// TwinCAT 3 PLC project SQLDemo
// ProgramVersion: 3.1.4026.22
// libraries:
//   Tc2_Standard, * (Beckhoff Automation GmbH)
//   Tc2_System, * (Beckhoff Automation GmbH)
//   Tc2_Utilities, * (Beckhoff Automation GmbH)
//   Tc3_Database, * (Beckhoff Automation GmbH)
//   Tc3_EventLogger, * (Beckhoff Automation GmbH)
// project tree:
//   DUTs/ ST_DbRecord.TcDUT
//   GVLs/ GVL_DB.TcGVL
//   / PlcTask.TcTTO
//   POUs/ FB_SqlLogger.TcPOU, MAIN.TcPOU
// real-time tasks:
//   TASK PlcTask: cycle T#10ms, priority 20, ADS port 350

CONFIGURATION SQLDemo
    RESOURCE PLC ON TwinCAT3
        TASK PlcTask(INTERVAL := T#10ms, PRIORITY := 21);
        PROGRAM MAIN WITH PlcTask : MAIN;
    END_RESOURCE
END_CONFIGURATION

// ---- DUTs/ST_DbRecord.TcDUT
// One row returned by a SELECT from the ds table
TYPE ST_DbRecord : STRUCT
  id        : DINT;
  timestamp : DT;
  value     : REAL;
END_STRUCT
END_TYPE

// ---- GVLs/GVL_DB.TcGVL
{attribute 'qualified_only'}
VAR_GLOBAL CONSTANT
  // Must match the hDBID configured in the TwinCAT Database Server (TF6420)
  DB_ID           : UDINT := 1;
  C_MaxSelectRows : UDINT := 1000;
END_VAR
VAR_GLOBAL
  arrResults   : ARRAY[1..1000] OF ST_DbRecord;
  nResultCount : UDINT;
  bWriteError  : BOOL;
END_VAR

// ---- POUs/MAIN.TcPOU
PROGRAM MAIN
VAR
  // --- System time (used by every FB_SqlLogger) ---
  fbLocalSystemTime : FB_LocalSystemTime;

  // --- Sensor values: replace these with your real signal variables ---
  rTemperature : REAL := 22.5;   // id=1
  rHumidity    : REAL := 55.0;   // id=2
  rSpeed       : REAL := 1450.0; // id=3

  // --- One logger per channel ---
  fbLogTemp  : FB_SqlLogger;
  fbLogHumid : FB_SqlLogger;
  fbLogSpeed : FB_SqlLogger;

  // --- Read back: set bSelect := TRUE to fetch the last 1000 rows ---
  fbSelectDb     : FB_SQLDatabaseEvt(sNetID := '', tTimeout := T#30S);
  fbSelectCmd    : FB_SQLCommandEvt(sNetID := '', tTimeout := T#30S);
  fbSelectResult : FB_SQLResultEvt(sNetID := '', tTimeout := T#30S);
  sSelectCmd     : STRING(255) := 'SELECT id, timestamp, value FROM ds ORDER BY timestamp DESC LIMIT 1000';
  bSelect        : BOOL;
  bSelectBusy    : BOOL;
  bSelectError   : BOOL;
  nSelectState   : INT; // 0=idle,1=connect,2=createCmd,3=execute,4=read,5=disconnect
  ipSelectResult : Tc3_EventLogger.I_TcMessage;
END_VAR

// --- System time ---
fbLocalSystemTime(bEnable := TRUE);

// --- Write: log each channel on its own interval ---
fbLogTemp(
  id           := 1,
  rValue       := rTemperature,
  nIntervalSec := 10,
  nDbHandle    := GVL_DB.DB_ID,
  stSystemTime := fbLocalSystemTime.systemTime);

fbLogHumid(
  id           := 2,
  rValue       := rHumidity,
  nIntervalSec := 10,
  nDbHandle    := GVL_DB.DB_ID,
  stSystemTime := fbLocalSystemTime.systemTime);

fbLogSpeed(
  id           := 3,
  rValue       := rSpeed,
  nIntervalSec := 10,
  nDbHandle    := GVL_DB.DB_ID,
  stSystemTime := fbLocalSystemTime.systemTime);

// Aggregate write errors for monitoring
GVL_DB.bWriteError := fbLogTemp.bError OR fbLogHumid.bError OR fbLogSpeed.bError;

// --- Read: triggered by setting bSelect := TRUE (e.g. from HMI or Watch window) ---
CASE nSelectState OF

  0: // Idle – waiting for trigger
    IF bSelect THEN
      nSelectState := 1;
    END_IF

  1: // Open connection
    IF fbSelectDb.Connect(GVL_DB.DB_ID) THEN
      ipSelectResult := fbSelectDb.ipTcResult;
      IF fbSelectDb.bError THEN
        bSelectError := TRUE;
        bSelect      := FALSE;
        nSelectState := 5;
      ELSE
        nSelectState := 2;
      END_IF
    END_IF

  2: // Bind command object
    IF fbSelectDb.CreateCmd(ADR(fbSelectCmd)) THEN
      ipSelectResult := fbSelectDb.ipTcResult;
      IF fbSelectDb.bError THEN
        bSelectError := TRUE;
        bSelect      := FALSE;
        nSelectState := 5;
      ELSE
        nSelectState := 3;
      END_IF
    END_IF

  3: // Execute SELECT and link result FB
    IF fbSelectCmd.ExecuteDataReturn(ADR(sSelectCmd), SIZEOF(sSelectCmd), ADR(fbSelectResult)) THEN
      ipSelectResult := fbSelectCmd.ipTcResult;
      IF fbSelectCmd.bError THEN
        bSelectError := TRUE;
        bSelect      := FALSE;
        nSelectState := 5;
      ELSE
        nSelectState := 4;
      END_IF
    END_IF

  4: // Read result rows into arrResults
    IF fbSelectResult.Read(0, GVL_DB.C_MaxSelectRows,
                           ADR(GVL_DB.arrResults), SIZEOF(GVL_DB.arrResults),
                           FALSE, TRUE) THEN
      ipSelectResult := fbSelectResult.ipTcResult;
      IF fbSelectResult.bError THEN
        bSelectError := TRUE;
      ELSE
        bSelectError          := FALSE;
        GVL_DB.nResultCount  := fbSelectResult.nDataCount;
      END_IF
      bSelect      := FALSE;
      nSelectState := 5;
    END_IF

  5: // Disconnect and return to idle
    IF fbSelectDb.Disconnect() THEN
      nSelectState := 0;
    END_IF

END_CASE

bSelectBusy := nSelectState <> 0;

END_PROGRAM

// ---- POUs/FB_SqlLogger.TcPOU
// Logs a single REAL value to a database table at a configurable cyclic interval.
// The DB timestamp is generated by MySQL (DEFAULT CURRENT_TIMESTAMP), so no
// system-time formatting is required here.
//
// Required MySQL table:
//   CREATE TABLE ds (
//     id        INT            NOT NULL,
//     timestamp DATETIME       NOT NULL DEFAULT CURRENT_TIMESTAMP,
//     value     FLOAT          NOT NULL
//   );
//
// Tc3_Database SQL Expert Mode: on first call the FB connects to the database
// and initialises a persistent FB_SQLCommandEvt. Subsequent inserts reuse the
// same open connection (states 0-1 run once; state 2 is the steady-state loop).
FUNCTION_BLOCK FB_SqlLogger
VAR_INPUT
  id           : DINT;           // Channel ID written to the 'id' column
  rValue       : REAL;           // Value to log
  nIntervalSec : INT := 10;      // How often to write (seconds)
  sTableName   : STRING := 'ds'; // Target table name
  nDbHandle    : UDINT;     // Database handle (configured in TF6420)
  stSystemTime : TIMESTRUCT;     // Pass fbLocalSystemTime.systemTime here
END_VAR
VAR_OUTPUT
  bBusy      : BOOL;
  bError     : BOOL;
  ipTcResult : Tc3_EventLogger.I_TcMessage;
END_VAR
VAR
  fbSqlDb        : FB_SQLDatabaseEvt(sNetID := '', tTimeout := T#10S);
  fbSqlCmd       : FB_SQLCommandEvt(sNetID := '', tTimeout := T#10S);
  rtrigSecond    : R_TRIG;
  wLastSecond    : WORD;
  nSecondCounter : INT;
  sInsertCmd     : STRING(255);
  bTrigInsert    : BOOL;
  nState         : INT; // 0=connecting, 1=createCmd, 2=ready, 3=executing, 255=error
  tonRetry : TON;
END_VAR

// Timing: count elapsed seconds and arm the insert trigger
rtrigSecond(CLK := stSystemTime.wSecond <> wLastSecond);
IF rtrigSecond.Q THEN
  wLastSecond := stSystemTime.wSecond;
  nSecondCounter := nSecondCounter + 1;
  IF nSecondCounter >= nIntervalSec THEN
    nSecondCounter := 0;
    // Build: INSERT INTO ds(id,value) VALUES (1,22.5)
    sInsertCmd := CONCAT('INSERT INTO ',
                  CONCAT(sTableName,
                  CONCAT('(id,value) VALUES (',
                  CONCAT(DINT_TO_STRING(id),
                  CONCAT(',',
                  CONCAT(REAL_TO_STRING(rValue), ')'))))));
    IF nState = 2 THEN // only arm when the connection is ready
      bTrigInsert := TRUE;
    END_IF
  END_IF
END_IF

// ── State machine ─────────────────────────────────────────────────────────────
CASE nState OF

  0: // Open connection to the configured database
    bBusy := TRUE;
    IF fbSqlDb.Connect(GVL_DB.DB_ID) THEN
      ipTcResult := fbSqlDb.ipTcResult;
      IF fbSqlDb.bError THEN
        bError := TRUE;
        nState := 255;
      ELSE
        nState := 1;
      END_IF
    END_IF

  1: // Bind a command object to the open connection
    IF fbSqlDb.CreateCmd(ADR(fbSqlCmd)) THEN
      ipTcResult := fbSqlDb.ipTcResult;
      IF fbSqlDb.bError THEN
        bError := TRUE;
        nState := 255;
      ELSE
        bError := FALSE;
        nState := 2;
      END_IF
    END_IF

  2: // Ready – waiting for the next insert trigger
    bBusy := FALSE;
    IF bTrigInsert THEN
      bTrigInsert := FALSE;
      nState := 3;
    END_IF

  3: // Execute the INSERT command asynchronously
    bBusy := TRUE;
    IF fbSqlCmd.Execute(ADR(sInsertCmd), SIZEOF(sInsertCmd)) THEN
      ipTcResult := fbSqlCmd.ipTcResult;
      bError := fbSqlCmd.bError;
      nState := 2; // return to ready regardless of outcome
    END_IF

  255: // Permanent error – connection or command initialisation failed
	  bBusy  := FALSE;
	  bError := TRUE;
	  tonRetry(IN := TRUE, PT := T#10S);
	  IF tonRetry.Q THEN
		tonRetry(IN := FALSE);
		bError := FALSE;
		nState := 0;  // retry connect
	  END_IF

END_CASE

END_FUNCTION_BLOCK
